Staubli VAL3: TCPConnect.pgx

program TCPConnect()
begin

  //there's nothing like client.connect in val3 socket...it's the os to handle this stuff when you try to write something!

end
